// Block: A04_DEBUG

DATA_BLOCK A04_DEBUG
VERSION : 0.1
   NON_RETAIN
   VAR
      Force_Sinamics_Infeed_ON : Bool;
      Force_Sinamics_Drives_CtrlSafe : Bool;
      Forse_Contactors_CtrlSafe : Bool;
      LsStratoDepositato : Bool;
      CIn_Manager_DEBUG : Struct
         PareggiatoreTesta : Struct
            Ax : Positioning_EPOS_Machine_COut;
         END_STRUCT;
         PareggiatoreCoda : Struct
            Ax : Positioning_EPOS_Machine_COut;
         END_STRUCT;
         Spalle : Struct
            Testa : Struct
               Ax : Positioning_DOL_Machine_COut;
            END_STRUCT;
            Coda : Struct
               Ax : Positioning_DOL_Machine_COut;
            END_STRUCT;
         END_STRUCT;
         Spintore : Struct
            Vrt : ValveMachine_COut;
            Orz : ValveMachine_COut;
         END_STRUCT;
         TraslazioneStrato : Struct
            Ax_Testa : Positioning_EPOS_Machine_COut;
            Ax_Coda : Positioning_EPOS_Machine_COut;
            Manip_Sostegno : ValveMachine_COut;
            Manip_Pareggiatore : ValveMachine_COut;
            SostegnoVrt : ValveMachine_COut;
         END_STRUCT;
         Sollevamento : Struct
            Ax_Testa : Positioning_DOL_Machine_COut;
            Ax_Coda : Positioning_DOL_Machine_COut;
         END_STRUCT;
         Sostegno : Struct
            Testa : Struct
               Ax : Positioning_DOL_Machine_COut;
               Paletto : Struct
                  CtrlSafe : Bool;
                  Standstill : Bool;
                  Rest_CheckNext : Bool;
                  Work_CheckNext : Bool;
                  Pos : Int;
                  RestPosition : Bool;
               END_STRUCT;
            END_STRUCT;
            Coda : Struct
               Ax : Positioning_DOL_Machine_COut;
               Paletto : Struct
                  CtrlSafe : Bool;
                  Standstill : Bool;
                  Rest_CheckNext : Bool;
                  Work_CheckNext : Bool;
                  Pos : Int;
                  RestPosition : Bool;
               END_STRUCT;
            END_STRUCT;
         END_STRUCT;
         Navetta : Struct
            ReadyToRecive : Bool;
            OutOfWorkspace : Bool;
            InPosizioneDiDeposito : Bool;
            RequestDeposito : Bool;
         END_STRUCT;
      END_STRUCT;
      CIn_Manager04_Debug : Struct
         Navetta : Struct
            Testa : Struct
               Ax : Positioning_DOL_Machine_COut;
               PalettiEsterni : ValveMachine_COut;
               PalettiInterni : ValveMachine_COut;
            END_STRUCT;
            Coda : Struct
               Ax : Positioning_DOL_Machine_COut;
               PalettiEsterni : ValveMachine_COut;
               PalettiInterni : ValveMachine_COut;
            END_STRUCT;
            Cumulativo : Struct
               PalettiEsterni : ValveMachine_COut;
               PalettiInterni : ValveMachine_COut;
            END_STRUCT;
         END_STRUCT;
         Sollevamento : Struct
            ReadyToDrop : Bool;
         END_STRUCT;
         Antiribaltamento : Struct
            Work : Bool;
            Rest : Bool;
         END_STRUCT;
      END_STRUCT;
      Beams_Data : Prod_Beam_Data;
      O_ID : Int;
   END_VAR

BEGIN
   // No initialization required
END_DATA_BLOCK
